{attribute 'qualified_only'}
{attribute 'strict'}
{attribute 'to_string'}
TYPE ENUM_Schunk :

(
	Init := 0,
	Undefined,
	Error,
	Reset,
	Stop,
	Ready,//Wait for command
	Homing,
	SetPosition,
	MoveAbsolute,
	MoveRelative
);	
	
END_TYPE

(* stored: Version 1.1.0.1, ProductVersion 3.1.4024.11
   DUT ENUM_Schunk: Id {4852b753-45bc-411e-a7d3-32a9d1cfab37} *)
